Yaskawa INFORM job: KRIS1A.JBI

/JOB
//NAME KRIS1A
///FOLDERNAME X4
//POS
///NPOS 161,161,159,7,0,0
///TOOL 0
///POSTYPE PULSE
///PULSE
C00000=-15579,-90125,-112680,751,85832,86751
C00001=112118,-87719,-111704,295,86466,-7981
C00002=112804,-79721,-69104,72,64358,-7781
C00003=115139,-78813,-67219,-786,63674,-6908
C00004=115139,-78456,-66016,-789,63117,-6905
C00005=115139,-78780,-67104,-787,63620,-6908
C00006=114295,-93268,-73076,-493,59845,-7207
C00007=115346,-91281,-70266,-899,59147,-6796
C00008=115425,-89696,-69639,-926,59575,-6770
C00009=114013,-96528,-75756,-385,59817,-7318
C00010=112176,-79610,-68801,301,64230,-8016
C00011=111826,-77700,-66544,429,63826,-8147
C00012=111826,-77414,-65561,430,63368,-8149
C00013=112189,-78969,-67115,296,63524,-8012
C00014=110981,-94268,-73476,769,59585,-8491
C00015=111195,-90668,-69679,691,59097,-8412
C00016=111340,-88986,-69006,634,59545,-8354
C00017=110917,-95978,-76175,788,60368,-8510
C00018=98905,-94426,-81055,5125,64609,-12947
C00019=104248,-50126,-59827,871,84915,-31292
C00020=110771,-18155,-40833,-2727,97609,-44192
C00021=111360,-18636,-39123,-2768,96333,-43971
C00022=111360,-18738,-38396,-2766,95833,-43962
C00023=110217,-18316,-38887,-2668,96314,-44350
C00024=110620,-19725,-39043,-2697,95701,-44202
C00025=110670,-19738,-39055,-2703,95699,-44187
C00026=109565,-18053,-39144,-2612,96586,-44572
C00027=114086,43998,16856,-2992,94166,-43015
C00028=114053,43978,17325,-2992,93865,-43021
C00029=114053,43945,17976,-2992,93449,-43011
C00030=113191,44226,17588,-2916,93800,-43307
C00031=113191,44191,18270,-2913,93364,-43296
C00032=113504,44097,18169,-2941,93388,-43192
C00033=113191,44297,16563,-2919,94467,-43322
C00034=95546,58384,35854,30061,98673,-46154
C00035=95582,58774,36295,30055,98599,-46160
C00036=123577,27205,-10716,19125,86619,-21364
C00037=146491,35264,3200,11924,78186,-14764
C00038=139465,39684,6918,23498,85006,-10799
C00039=143221,41856,17232,31724,78736,-2144
C00040=143777,45964,21760,32091,77889,-1898
C00041=143777,45970,22332,32127,77590,-1984
C00042=143777,45964,21760,32091,77889,-1898
C00043=144048,47864,23803,32049,77548,-1889
C00044=143777,45964,21760,32091,77889,-1898
C00045=140515,27172,13,30557,79503,260
C00046=127712,47757,18303,22708,83382,-6719
C00047=131160,50524,19335,14874,81362,-8697
C00048=131524,51962,21137,14784,80938,-8621
C00049=131524,51834,22237,14811,80220,-8709
C00050=131524,51962,21137,14784,80938,-8621
C00051=131412,54587,24038,14832,80535,-8708
C00052=124540,58684,30159,20118,82239,-15737
C00053=124540,58684,30159,20118,82239,-15737
C00054=126244,67376,38231,22849,84013,-19503
C00055=125634,64122,36548,22992,83592,-19805
C00056=124813,61662,33823,22854,83980,-19602
C00057=136187,52210,23726,20634,82490,-16225
C00058=138691,53299,30320,37349,84215,-2442
C00059=138736,52471,34602,46175,82339,-1039
C00060=124737,44137,16346,44293,94212,-2593
C00061=119692,30389,-7142,25705,97127,-4865
C00062=118955,27408,-15020,17592,99243,-80195
C00063=125200,-2101,-32741,15880,81610,-85840
C00064=134088,-16964,-41109,182,70766,-85347
C00065=127415,46663,16862,1950,67717,-87809
C00066=121903,36391,497,16998,81593,-86950
C00067=125298,-36844,-66213,15778,84239,-85470
C00068=119205,-70443,-76936,24876,74885,-88203
C00069=118806,-67965,-71783,25211,73277,-88701
C00070=119684,40726,11380,24463,77277,-87514
C00071=126391,-52827,-68733,22124,76579,-85223
C00072=119612,-43604,-61782,23842,90714,-84840
C00073=150919,-31098,-53968,16672,84728,-75038
C00074=142912,-38104,-51044,32938,76311,-77903
C00075=131483,-69573,-74262,36162,79312,-81611
C00076=134129,-100468,-92829,36100,74575,-82089
C00077=-15579,-90125,-112680,751,85832,86751
C00078=-15579,-90125,-112680,751,85832,86751
C00079=-15579,-90125,-112677,751,85834,86750
C00080=-3695,-78746,-107796,-19987,71227,-76789
C00081=-15579,-90125,-112677,751,85834,86750
C00082=69723,-89114,-112269,359,86097,-2011
C00083=103224,-63598,-76709,4432,93708,-9007
C00084=100150,-62593,-71932,4790,91465,-10109
C00085=102335,-62307,-70304,4519,90489,-9417
C00086=102335,-62333,-69297,4519,89858,-9438
C00087=102335,-62306,-70332,4519,90507,-9413
C00088=99769,-80336,-79078,4826,86783,-10413
C00089=98266,-88378,-78396,6942,76534,-11334
C00090=98474,-87229,-77918,6891,76813,-11243
C00091=99558,-93232,-83375,6670,76995,-10858
C00092=70996,-48839,-62917,11636,90314,-19604
C00093=69525,-45287,-58669,11857,89748,-20153
C00094=69525,-45355,-57854,11856,89224,-20204
C00095=69525,-45284,-58714,11860,89779,-20150
C00096=64327,-57195,-66086,12620,89001,-21989
C00097=64937,-55938,-62941,12533,87648,-21918
C00098=65630,-54449,-62112,12434,87792,-21669
C00099=64207,-57448,-65984,12639,88833,-22049
C00100=106021,-71460,-78290,5261,84540,-8299
C00101=112603,-50924,-67434,3896,88035,39850
C00102=99785,-49787,-63878,14924,89163,36712
C00103=99827,-50120,-62714,14916,88297,36622
C00104=99827,-50195,-61812,14916,87722,36551
C00105=99827,-50144,-62447,14916,88126,36600
C00106=101735,-51128,-63015,14585,87637,37193
C00107=101608,-51204,-62348,14606,87222,37100
C00108=101075,-50939,-62194,14699,87359,36934
C00109=102139,-51368,-63677,14510,87842,37354
C00110=99650,-48435,-63078,14947,89385,36690
C00111=99972,-48773,-61841,14889,88425,36682
C00112=99972,-48836,-61171,14890,87997,36629
C00113=99984,-48651,-62050,14887,88610,36709
C00114=102057,-49715,-62671,14526,88085,37352
C00115=101809,-49682,-61617,14570,87514,37201
C00116=101235,-49486,-61523,14671,87658,37023
C00117=101817,-49661,-62901,14567,88291,37295
C00118=100331,-60546,-70178,19462,73070,35082
C00119=112110,-11200,-31080,-21080,73268,936
C00120=112400,17878,-3446,-21379,75013,1233
C00121=111590,19523,-1910,-21129,74714,991
C00122=111590,19505,-1171,-21171,74277,1069
C00123=111547,19542,-1905,-21114,74709,976
C00124=111586,21327,-236,-21132,74618,1008
C00125=111547,19542,-1905,-21114,74709,976
C00126=112862,2673,-16978,-21482,75612,1293
C00127=115448,-25762,-50567,-21911,81920,1062
C00128=115448,-26322,-48444,-21988,80436,1335
C00129=82803,-6073,-29763,-10236,73084,-8971
C00130=79384,-350,-31136,-8698,76436,-10385
C00131=79572,10395,-14436,-8965,71755,-9979
C00132=79534,10356,-13587,-8976,71217,-9951
C00133=79572,10395,-14436,-8965,71755,-9979
C00134=79918,12066,-12957,-9108,71739,-9858
C00135=79284,8995,-16143,-8832,72049,-10102
C00136=90478,36773,12863,-10350,74792,593
C00137=94157,33011,8641,-3718,74256,-1986
C00138=94889,36373,12557,5370,72876,-270
C00139=91513,44429,23385,15929,70108,-695
C00140=94206,50619,32489,25830,69108,-1135
C00141=99622,24209,5008,27862,67795,3286
C00142=101698,-3167,-21798,-5919,61845,73
C00143=117691,-82819,-72183,-15832,54407,7355
C00144=136102,-94056,-81974,-24248,59304,-21802
C00145=127300,-9107,-38878,-10715,73507,-75725
C00146=127883,-10256,-28747,-11426,66877,-74900
C00147=125820,57665,36060,-10904,61708,-75162
C00148=125724,45909,15983,-10333,67906,-75775
C00149=151418,-11051,-30715,-39158,77226,-70934
C00150=166637,-124928,-92814,-37840,63906,-58834
C00151=182097,-119423,-82240,-42095,69399,-53697
C00152=148901,-14656,-27686,-35717,72453,-69897
C00153=152618,-101160,-84187,-32865,63932,-65185
C00154=146642,-96347,-88741,-9688,84313,-74893
C00155=146358,-95495,-85194,-9676,82559,-74858
C00156=129145,-102178,-86219,-14985,78455,-80586
C00157=126274,-93471,-76691,-31678,80491,-81832
C00158=136204,-90113,-81071,-25794,88530,-79839
C00159=135637,-91176,-85093,-22103,89594,-80119
C00160=-3208,-93475,-86259,-2679,87523,-79016
BC00000=99,526410,1075081
BC00001=171737,515230,306420
BC00002=55459,454786,199131
BC00003=55459,454786,199131
BC00004=55459,454786,199131
BC00005=55459,454786,199131
BC00006=55459,454786,199131
BC00007=55459,454786,199131
BC00008=55459,454786,199131
BC00009=55459,454786,199131
BC00010=108304,454786,199131
BC00011=108304,454786,199131
BC00012=108304,454786,199131
BC00013=108304,454786,199131
BC00014=108304,454786,199131
BC00015=108304,454786,199131
BC00016=108304,454786,199131
BC00017=108304,454786,199131
BC00018=108304,454786,199131
BC00019=108304,454786,199131
BC00020=108304,454786,199131
BC00021=108304,454786,199131
BC00022=108304,454786,199131
BC00023=108304,454786,199131
BC00024=108304,454786,199131
BC00025=108304,454786,199131
BC00026=108304,454786,199131
BC00027=108304,440546,199131
BC00028=108304,440546,199131
BC00029=108304,440546,199131
BC00030=108304,440546,199131
BC00031=108304,440546,199131
BC00032=108304,440546,199130
BC00033=108304,440546,199131
BC00034=108304,440546,199131
BC00035=108304,440546,199131
BC00036=153886,383281,124194
BC00037=174583,383281,124194
BC00038=163957,383281,124194
BC00039=168122,383282,124193
BC00040=170139,383282,124190
BC00041=170139,383282,124190
BC00042=170139,383282,124190
BC00043=170139,383282,124190
BC00044=170139,383282,124190
BC00045=170139,383282,124190
BC00046=146661,383281,124193
BC00047=154148,383281,124194
BC00048=154148,383281,124194
BC00049=154148,383281,124194
BC00050=154148,383281,124194
BC00051=154148,383281,124194
BC00052=140502,383282,124191
BC00053=140502,383282,124191
BC00054=154149,383281,124191
BC00055=154149,383281,124191
BC00056=141565,383281,124189
BC00057=154149,383281,124188
BC00058=154152,383279,124187
BC00059=154149,383281,124191
BC00060=139202,383281,124191
BC00061=134656,383281,124191
BC00062=136731,381659,124191
BC00063=152069,383281,124191
BC00064=150142,383281,124191
BC00065=138256,383281,124191
BC00066=136697,383281,124191
BC00067=170077,383281,124191
BC00068=170077,446955,124191
BC00069=170077,446955,124191
BC00070=170077,446955,124191
BC00071=170077,446955,124191
BC00072=170077,446955,124191
BC00073=170077,446955,124191
BC00074=170077,446955,124191
BC00075=170077,446955,124191
BC00076=170077,446955,124191
BC00077=99,526410,1075081
BC00078=99,526410,1075081
BC00079=99,526409,1075080
BC00080=199448,515539,1075137
BC00081=141247,502779,337681
BC00082=222419,439021,164840
BC00083=279909,439021,164840
BC00084=279909,439021,164840
BC00085=279909,439021,164840
BC00086=279909,439021,164840
BC00087=279909,439021,164840
BC00088=279909,439021,164840
BC00089=279909,439021,164840
BC00090=279909,439021,164840
BC00091=279909,439021,164840
BC00092=279909,439021,164840
BC00093=279909,439021,164840
BC00094=279909,439021,164840
BC00095=279909,439021,164840
BC00096=279909,439021,164840
BC00097=279909,439021,164840
BC00098=279909,439021,164840
BC00099=279909,439021,164840
BC00100=279909,439021,164840
BC00101=279909,439021,164840
BC00102=279909,439021,164840
BC00103=279909,439021,164840
BC00104=279909,439021,164840
BC00105=279909,439021,164840
BC00106=279909,439021,164840
BC00107=279909,439021,164840
BC00108=279909,439021,164840
BC00109=279909,439021,164840
BC00110=279909,350395,164840
BC00111=279909,350395,164840
BC00112=279909,350395,164840
BC00113=279909,350395,164840
BC00114=279909,350395,164840
BC00115=279909,350395,164840
BC00116=279909,350395,164840
BC00117=279909,350395,164840
BC00118=279909,350395,164840
BC00119=279909,350395,164840
BC00120=279909,355371,164840
BC00121=279909,355371,164840
BC00122=279909,355371,164840
BC00123=279909,355371,164840
BC00124=279909,355371,164840
BC00125=279909,355371,164840
BC00126=279909,355371,164840
BC00127=279909,355371,164840
BC00128=279909,427919,164840
BC00129=247234,427919,164840
BC00130=278465,363509,138086
BC00131=278465,363509,138086
BC00132=278465,363509,138086
BC00133=278465,363509,138086
BC00134=278465,363509,138086
BC00135=278465,363509,138086
BC00136=302650,395853,164837
BC00137=311944,395852,164836
BC00138=309501,395853,164836
BC00139=296323,395854,164837
BC00140=301591,395854,164837
BC00141=326424,395853,164837
BC00142=326424,395853,164837
BC00143=326424,395853,164837
BC00144=326424,395853,164837
BC00145=326424,395853,164837
BC00146=326869,395161,164261
BC00147=326869,395161,164261
BC00148=326869,395161,164261
BC00149=326869,395161,164261
BC00150=326869,395161,164261
BC00151=326869,395161,164261
BC00152=326869,395161,164261
BC00153=326869,395161,164261
BC00154=326869,395161,164261
BC00155=326869,395161,164261
BC00156=326869,395161,164261
BC00157=326869,395161,164260
BC00158=326869,395161,164259
BC00159=326869,452441,213700
BC00160=87826,515074,1040939
EC00000=-798157,-183832
EC00001=-798154,-183834
EC00002=-798154,-183834
EC00003=-798154,-183834
EC00004=-798154,-183834
EC00005=-798154,-183834
EC00006=-798154,-183834
EC00007=-798154,-183834
EC00008=-798154,-183834
EC00009=-798154,-183834
EC00010=-798154,-183834
EC00011=-798154,-183834
EC00012=-798154,-183834
EC00013=-798154,-183834
EC00014=-798154,-183834
EC00015=-798154,-183834
EC00016=-798154,-183834
EC00017=-798154,-183834
EC00018=-798154,-183834
EC00019=-798154,-183834
EC00020=-798154,-183834
EC00021=-798154,-183834
EC00022=-798154,-183834
EC00023=-798154,-183834
EC00024=-798154,-183834
EC00025=-798154,-183834
EC00026=-798154,-183834
EC00027=-798154,-183834
EC00028=-798154,-183834
EC00029=-798154,-183834
EC00030=-798154,-183834
EC00031=-798154,-183834
EC00032=-798153,-183834
EC00033=-798154,-183834
EC00034=-798154,-183834
EC00035=-798154,-183834
EC00036=-798154,-183834
EC00037=-798154,-183834
EC00038=-798154,-183834
EC00039=-798153,-183835
EC00040=-798152,-183835
EC00041=-798152,-183835
EC00042=-798152,-183835
EC00043=-798152,-183835
EC00044=-798152,-183835
EC00045=-798152,-183835
EC00046=-798154,-183834
EC00047=-798154,-183834
EC00048=-798154,-183834
EC00049=-798154,-183834
EC00050=-798154,-183834
EC00051=-798154,-183834
EC00052=-798151,-183838
EC00053=-798151,-183838
EC00054=-798151,-183835
EC00055=-798151,-183835
EC00056=-798151,-183835
EC00057=-798153,-183834
EC00058=-798153,-183834
EC00059=-798153,-183834
EC00060=-798153,-183834
EC00061=-798153,-183834
EC00062=-798153,-183834
EC00063=-798153,-183834
EC00064=-798153,-183834
EC00065=-798153,-183834
EC00066=-798153,-183834
EC00067=-798153,-183834
EC00068=-798153,-183834
EC00069=-798153,-183834
EC00070=-798153,-183834
EC00071=-798153,-183834
EC00072=-798153,-183834
EC00073=-798153,-183834
EC00074=-798153,-183834
EC00075=-798157,-183832
EC00076=-93266,-194312
EC00077=-184298,-1289476
EC00078=-798157,-1296784
EC00079=-798157,-1296784
EC00080=-798156,-1296783
EC00081=-798156,-1296783
EC00082=-798156,-1296783
EC00083=-798156,-1296783
EC00084=-798156,-1296783
EC00085=-798156,-1296783
EC00086=-798156,-1296783
EC00087=-798156,-1296783
EC00088=-798156,-1296783
EC00089=-798156,-1296783
EC00090=-798156,-1296783
EC00091=-798156,-1296783
EC00092=-798156,-1296783
EC00093=-798156,-1296783
EC00094=-798156,-1296783
EC00095=-798156,-1296783
EC00096=-798156,-1296783
EC00097=-798156,-1296783
EC00098=-798156,-1296783
EC00099=-798156,-1296783
EC00100=-798156,-1296783
EC00101=-798156,-1296783
EC00102=-798156,-1296783
EC00103=-798156,-1296783
EC00104=-798156,-1296783
EC00105=-798156,-1296783
EC00106=-798156,-1296783
EC00107=-798156,-1296783
EC00108=-798156,-1296783
EC00109=-798156,-1296783
EC00110=-798156,-1296783
EC00111=-798156,-1296783
EC00112=-798156,-1296783
EC00113=-798156,-1296783
EC00114=-798156,-1296783
EC00115=-798156,-1296783
EC00116=-798156,-1296783
EC00117=-798156,-1296783
EC00118=-798156,-1296783
EC00119=-798156,-1296783
EC00120=-798156,-1296783
EC00121=-798156,-1296783
EC00122=-798156,-1296783
EC00123=-798156,-1296783
EC00124=-798156,-1296783
EC00125=-798156,-1296783
EC00126=-798156,-1296783
EC00127=-798156,-1296783
EC00128=-798156,-1296783
EC00129=-798156,-1296783
EC00130=-798156,-1296783
EC00131=-798156,-1296783
EC00132=-798156,-1296783
EC00133=-798156,-1296783
EC00134=-798155,-1296782
EC00135=-798154,-1296780
EC00136=-798153,-1296781
EC00137=-798154,-1296781
EC00138=-798154,-1296781
EC00139=-798155,-1296782
EC00140=-798155,-1296782
EC00141=-798155,-1296782
EC00142=-798155,-1296782
EC00143=-798155,-1296782
EC00144=-798155,-1296782
EC00145=-798155,-1296782
EC00146=-798155,-1296782
EC00147=-798155,-1296782
EC00148=-798155,-1296782
EC00149=-798155,-1296782
EC00150=-798155,-1296782
EC00151=-798155,-1296782
EC00152=-798155,-1296782
EC00153=-798155,-1296782
EC00154=-798155,-1296782
EC00155=-798154,-1296781
EC00156=-798154,-1296780
EC00157=-798154,-1296780
EC00158=-798154,-1287204
///POSTYPE BASE
///RECTAN
///RCONF 0,0,0,0,1,0,0,0,0,0,0,0,0,0,0,0,0,0,0,0,0,0,0,0
P00006=2.006,1.622,-0.565,0.0000,0.0000,0.0000
P00021=0.073,2.058,-0.109,0.0000,0.0000,0.0000
P00022=2.006,1.622,-0.565,0.0000,0.0000,0.0000
///RCONF 0,0,0,0,0,0,0,0,0,0,0,0,0,0,0,0,0,0,0,0,0,0,0,0
P00023=-2.957,-4.083,2.762,0.0000,0.0000,0.0000
P00024=-1.466,-0.226,-0.419,0.0000,0.0000,0.0000
P00025=3.643,0.007,-2.585,0.0000,0.0000,0.0000
P00026=2.644,0.055,-2.583,0.0000,0.0000,0.0000
//INST
///DATE 2024/11/13 16:42
///ATTR SC,RW
///GROUP1 RB1,BS1
///GROUP2 ST1
NOP
SFTOF3D
CALL JOB:CLEAN-R1_KM_NEW
MOVJ C00000 BC00000 VJ=100.00  +MOVJ EC00000 VJ=100.00
MOVJ C00001 BC00001 VJ=100.00  +MOVJ EC00001 VJ=100.00
MOVJ C00002 BC00002 VJ=100.00  +MOVJ EC00002 VJ=100.00
SMOVL C00003 BC00003 V=100.0  +MOVJ EC00003
SREFP 3 C00004 BC00004  +REFP EC00004
CALL JOB:SEARCH-R1-S13D
SET P023 P006
SFTON3D P023
SMOVL C00005 BC00005 V=133.3  +MOVJ EC00005
SMOVL C00006 BC00006 V=133.3  +MOVJ EC00006
SMOVL C00007 BC00007 V=133.3  +MOVJ EC00007
SREFP 3 C00008 BC00008  +REFP EC00008
CALL JOB:SEARCH-R1-S13D
SET P023 P006
SFTON3D P023
SMOVL C00009 BC00009 V=166.7  +MOVJ EC00009
SFTOF
SFTOF3D
SMOVL C00010 BC00010 V=250.0  +MOVJ EC00010
SMOVL C00011 BC00011 V=100.0  +MOVJ EC00011
SREFP 3 C00012 BC00012  +REFP EC00012
CALL JOB:SEARCH-R1-S13D
SET P024 P006
SFTON3D P024
SMOVL C00013 BC00013 V=133.3  +MOVJ EC00013
SMOVL C00014 BC00014 V=133.3  +MOVJ EC00014
SMOVL C00015 BC00015 V=133.3  +MOVJ EC00015
SREFP 3 C00016 BC00016  +REFP EC00016
CALL JOB:SEARCH-R1-S13D
SET P024 P006
SFTON3D P024
SMOVL C00017 BC00017 V=166.7  +MOVJ EC00017
SFTOF3D
MOVJ C00018 BC00018 VJ=100.00  +MOVJ EC00018 VJ=100.00
MOVJ C00019 BC00019 VJ=100.00  +MOVJ EC00019 VJ=100.00
MOVJ C00020 BC00020 VJ=100.00  +MOVJ EC00020 VJ=100.00
SMOVL C00021 BC00021 V=100.0  +MOVJ EC00021
SREFP 3 C00022 BC00022  +REFP EC00022
CALL JOB:SEARCH-R1-S13D
SET P025 P006
SFTON3D P025
SMOVL C00023 BC00023 V=100.0  +MOVJ EC00023
SMOVL C00024 BC00024 V=100.0  +MOVJ EC00024
SREFP 3 C00025 BC00025  +REFP EC00025
CALL JOB:SEARCH-R1-S13D
SET P025 P006
SFTON3D P025
SMOVL C00026 BC00026 V=100.0  +MOVJ EC00026
SFTOF3D
SFTOF
SMOVL C00027 BC00027 V=500.0  +MOVJ EC00027
SMOVL C00028 BC00028 V=100.0  +MOVJ EC00028
SREFP 3 C00029 BC00029  +REFP EC00029
CALL JOB:SEARCH-R1-S13D
SET P026 P006
SFTON3D P026
SMOVL C00030 BC00030 V=133.3  +MOVJ EC00030
SMOVL C00031 BC00031 V=100.0  +MOVJ EC00031
SREFP 3 C00032 BC00032  +REFP EC00032
CALL JOB:SEARCH-R1-S13D
SET P026 P006
SFTON3D P026
SMOVL C00033 BC00033 V=166.7  +MOVJ EC00033
SFTOF3D
SFTOF
SMOVL C00034 BC00034 V=500.0  +MOVJ EC00034
MOVJ C00035 BC00035 VJ=100.00  +MOVJ EC00035 VJ=100.00
MOVJ C00036 BC00036 VJ=100.00  +MOVJ EC00036 VJ=20.00
MOVJ C00037 BC00037 VJ=20.00  +MOVJ EC00037 VJ=20.00
MOVJ C00038 BC00038 VJ=20.00  +MOVJ EC00038 VJ=20.00
MOVJ C00039 BC00039 VJ=20.00  +MOVJ EC00039 VJ=20.00
SMOVL C00040 BC00040 V=100.0  +MOVJ EC00040
SREFP 3 C00041 BC00041  +REFP EC00041
CALL JOB:SEARCH-R1-S13D
SET P022 P006
SFTON3D P022
SMOVL C00042 BC00042 V=100.0  +MOVJ EC00042
SREFP 3 C00043 BC00043  +REFP EC00043
CALL JOB:SEARCH-R1-S13D
SET P022 P006
SFTON3D P022
SMOVL C00044 BC00044 V=100.0  +MOVJ EC00044
SFTOF3D
MOVL C00045 BC00045 V=500.0  +MOVJ EC00045 VJ=20.00
MOVL C00046 BC00046 V=500.0  +MOVJ EC00046 VJ=20.00
SMOVL C00047 BC00047 V=500.0  +MOVJ EC00047
SMOVL C00048 BC00048 V=100.0  +MOVJ EC00048
SREFP 3 C00049 BC00049  +REFP EC00049
CALL JOB:SEARCH-R1-S13D
SET P021 P006
SFTON3D P021
SMOVL C00050 BC00050 V=100.0  +MOVJ EC00050
SREFP 3 C00051 BC00051  +REFP EC00051
CALL JOB:SEARCH-R1-S13D
SET P021 P006
SFTON3D P021
SMOVL C00052 BC00052 V=100.0  +MOVJ EC00052
MACRO1 MJ#(0) ARGF21
SMOVL C00053 BC00053 V=250.0  +MOVJ EC00053
REFP 1 RB1 C00054 BC00054
REFP 2 RB1 C00055 BC00055
ARCON
SWVON WEV#(100)
SMOVL C00056 BC00056 V=8.3  +MOVJ EC00054
SFTON3D P022
SMOVL C00057 BC00057 V=8.3  +MOVJ EC00055
SMOVL C00058 BC00058 V=8.3  +MOVJ EC00056
SMOVL C00059 BC00059 V=8.3  +MOVJ EC00057
ARCOF
SWVOF
SFTOF
SFTOF3D
SMOVL C00060 BC00060 V=333.3  +MOVJ EC00058
SMOVL C00061 BC00061 V=666.7  +MOVJ EC00059
MOVJ C00062 BC00062 VJ=100.00  +MOVJ EC00060 VJ=20.00
MOVJ C00063 BC00063 VJ=70.00  +MOVJ EC00061 VJ=20.00
MACRO1 MJ#(0) ARGF20
SFTON3D P025
SMOVL C00064 BC00064 V=250.0  +MOVJ EC00062
ARCON
SFTON3D P026
SMOVL C00065 BC00065 V=7.5  +MOVJ EC00063
ARCOF
SWVOF
SFTOF3D
SFTOF
SMOVL C00066 BC00066 V=333.3  +MOVJ EC00064
SMOVL C00067 BC00067 V=666.7  +MOVJ EC00065
MACRO1 MJ#(0) ARGF14
SMOVL C00068 BC00068 V=500.0  +MOVJ EC00066
SFTON3D P025
SMOVL C00069 BC00069 V=166.7  +MOVJ EC00067
ARCON
SWVON WEV#(20)
SFTON3D P026
SMOVL C00070 BC00070 V=10.0  +MOVJ EC00068
ARCOF
SWVOF
SFTOF
SFTOF3D
SMOVL C00071 BC00071 V=333.3  +MOVJ EC00069
SFTON3D P024
SMOVL C00072 BC00072 V=166.7  +MOVJ EC00070
ARCON
SWVON WEV#(20)
SFTON3D P023
SMOVL C00073 BC00073 V=12.5  +MOVJ EC00071
SMOVL C00074 BC00074 V=12.5  +MOVJ EC00072
ARCOF
SWVOF
SFTOF
SFTOF3D
SMOVL C00075 BC00075 V=500.0  +MOVJ EC00073
SMOVL C00076 BC00076 V=1000.0  +MOVJ EC00074
MOVJ C00077 BC00077 VJ=100.00  +MOVJ EC00075 VJ=20.00
MOVJ C00078 BC00078 VJ=100.00  +MOVJ EC00076 VJ=100.00
MOVJ C00079 BC00079 VJ=100.00  +MOVJ EC00077 VJ=100.00
MOVJ C00080 BC00080 VJ=100.00  +MOVJ EC00078 VJ=100.00
'DRUGA STRONA
CALL JOB:CLEAN-R1_KM_NEW
MOVJ C00081 BC00081 VJ=100.00  +MOVJ EC00079 VJ=100.00
MOVJ C00082 BC00082 VJ=100.00  +MOVJ EC00080 VJ=100.00
MOVJ C00083 BC00083 VJ=100.00  +MOVJ EC00081 VJ=100.00
SFTOF3D
MOVJ C00084 BC00084 VJ=100.00  +MOVJ EC00082 VJ=100.00
SMOVL C00085 BC00085 V=166.7  +MOVJ EC00083
SREFP 3 C00086 BC00086  +REFP EC00084
CALL JOB:SEARCH-R1-S13D
SET P023 P006
SFTON3D P023
SMOVL C00087 BC00087 V=250.0  +MOVJ EC00085
SMOVL C00088 BC00088 V=250.0  +MOVJ EC00086
SMOVL C00089 BC00089 V=250.0  +MOVJ EC00087
SREFP 3 C00090 BC00090  +REFP EC00088
CALL JOB:SEARCH-R1-S13D
SET P023 P006
SFTON3D P023
SFTOF3D
SFTOF
SMOVL C00091 BC00091 V=250.0  +MOVJ EC00089
SMOVL C00092 BC00092 V=250.0  +MOVJ EC00090
SMOVL C00093 BC00093 V=250.0  +MOVJ EC00091
SREFP 3 C00094 BC00094  +REFP EC00092
CALL JOB:SEARCH-R1-S13D
SET P024 P006
SFTON3D P024
SMOVL C00095 BC00095 V=250.0  +MOVJ EC00093
SMOVL C00096 BC00096 V=250.0  +MOVJ EC00094
SMOVL C00097 BC00097 V=250.0  +MOVJ EC00095
SREFP 3 C00098 BC00098  +REFP EC00096
CALL JOB:SEARCH-R1-S13D
SET P024 P006
SFTON3D P024
SFTOF3D
SMOVL C00099 BC00099 V=250.0  +MOVJ EC00097
MOVJ C00100 BC00100 VJ=100.00  +MOVJ EC00098 VJ=100.00
MOVJ C00101 BC00101 VJ=100.00  +MOVJ EC00099 VJ=100.00
MOVJ C00102 BC00102 VJ=100.00  +MOVJ EC00100 VJ=100.00
SMOVL C00103 BC00103 V=250.0  +MOVJ EC00101
SREFP 3 C00104 BC00104  +REFP EC00102
CALL JOB:SEARCH-R1-S13D
SET P025 P006
SFTON3D P025
SMOVL C00105 BC00105 V=250.0  +MOVJ EC00103
SMOVL C00106 BC00106 V=250.0  +MOVJ EC00104
SMOVL C00107 BC00107 V=100.0  +MOVJ EC00105
SREFP 3 C00108 BC00108  +REFP EC00106
CALL JOB:SEARCH-R1-S13D
SET P025 P006
SFTON3D P025
SFTOF3D
SMOVL C00109 BC00109 V=100.0  +MOVJ EC00107
SMOVL C00110 BC00110 V=333.3  +MOVJ EC00108
SMOVL C00111 BC00111 V=250.0  +MOVJ EC00109
SREFP 3 C00112 BC00112  +REFP EC00110
CALL JOB:SEARCH-R1-S13D
SET P026 P006
SFTON3D P026
SMOVL C00113 BC00113 V=250.0  +MOVJ EC00111
SMOVL C00114 BC00114 V=250.0  +MOVJ EC00112
SMOVL C00115 BC00115 V=100.0  +MOVJ EC00113
SREFP 3 C00116 BC00116  +REFP EC00114
CALL JOB:SEARCH-R1-S13D
SET P026 P006
SFTON3D P026
SFTOF3D
SMOVL C00117 BC00117 V=250.0  +MOVJ EC00115
SMOVL C00118 BC00118 V=333.3  +MOVJ EC00116
MOVJ C00119 BC00119 VJ=20.00  +MOVJ EC00117 VJ=20.00
MOVJ C00120 BC00120 VJ=20.00  +MOVJ EC00118 VJ=20.00
SMOVL C00121 BC00121 V=250.0  +MOVJ EC00119
SREFP 3 C00122 BC00122  +REFP EC00120
CALL JOB:SEARCH-R1-S13D
SET P021 P006
SFTON3D P021
SMOVL C00123 BC00123 V=250.0  +MOVJ EC00121
SREFP 3 C00124 BC00124  +REFP EC00122
CALL JOB:SEARCH-R1-S13D
SET P021 P006
SFTON3D P021
SFTOF3D
SMOVL C00125 BC00125 V=250.0  +MOVJ EC00123
MOVL C00126 BC00126 V=250.0  +MOVJ EC00124 VJ=20.00
MOVL C00127 BC00127 V=333.3  +MOVJ EC00125 VJ=20.00
SMOVL C00128 BC00128 V=1000.0  +MOVJ EC00126
SMOVL C00129 BC00129 V=1000.0  +MOVJ EC00127
SMOVL C00130 BC00130 V=250.0  +MOVJ EC00128
SMOVL C00131 BC00131 V=250.0  +MOVJ EC00129
SREFP 3 C00132 BC00132  +REFP EC00130
CALL JOB:SEARCH-R1-S13D
SET P022 P006
SFTON3D P022
SMOVL C00133 BC00133 V=250.0  +MOVJ EC00131
SREFP 3 C00134 BC00134  +REFP EC00132
CALL JOB:SEARCH-R1-S13D
SET P022 P006
SFTOF3D
SMOVL C00135 BC00135 V=250.0  +MOVJ EC00133
MACRO1 MJ#(0) ARGF21
SFTON3D P022
SMOVL C00136 BC00136 V=250.0  +MOVJ EC00134
ARCON
SWVON WEV#(100)
SMOVL C00137 BC00137 V=8.3  +MOVJ EC00135
SMOVL C00138 BC00138 V=8.3  +MOVJ EC00136
SFTON3D P021
SMOVL C00139 BC00139 V=8.3  +MOVJ EC00137
SMOVL C00140 BC00140 V=8.3  +MOVJ EC00138
ARCOF
SFTOF3D
SWVOF
SMOVL C00141 BC00141 V=250.0  +MOVJ EC00139
SMOVL C00142 BC00142 V=500.0  +MOVJ EC00140
MOVJ C00143 BC00143 VJ=50.00  +MOVJ EC00141 VJ=20.00
MOVJ C00144 BC00144 VJ=100.00  +MOVJ EC00142 VJ=20.00
MOVJ C00145 BC00145 VJ=40.00  +MOVJ EC00143 VJ=20.00
MACRO1 MJ#(0) ARGF20
SFTON3D P025
SMOVL C00146 BC00146 V=133.3 PL=0  +MOVJ EC00144
ARCON
SFTON3D P026
SMOVL C00147 BC00147 V=6.7  +MOVJ EC00145
ARCOF
SWVOF
SFTOF3D
SMOVL C00148 BC00148 V=250.0  +MOVJ EC00146
SMOVL C00149 BC00149 V=500.0  +MOVJ EC00147
MACRO1 MJ#(0) ARGF14
SFTOF3D
SMOVL C00150 BC00150 V=500.0  +MOVJ EC00148
SFTOF
SFTON3D P025
SMOVL C00151 BC00151 V=250.0  +MOVJ EC00149
ARCON
SWVON WEV#(20)
SFTON3D P026
SMOVL C00152 BC00152 V=10.0  +MOVJ EC00150
ARCOF
SWVOF
SFTOF3D
SMOVL C00153 BC00153 V=333.3  +MOVJ EC00151
MOVL C00154 BC00154 V=250.0  +MOVJ EC00152 VJ=100.00
SFTON3D P023
SMOVL C00155 BC00155 V=250.0  +MOVJ EC00153
ARCON
SWVON WEV#(20)
SFTON3D P024
SMOVL C00156 BC00156 V=11.7  +MOVJ EC00154
SMOVL C00157 BC00157 V=11.7  +MOVJ EC00155
ARCOF
SWVOF
SFTOF
SMOVL C00158 BC00158 V=250.0  +MOVJ EC00156
MOVJ C00159 BC00159 VJ=100.00  +MOVJ EC00157 VJ=20.00
MOVJ C00160 BC00160 VJ=100.00  +MOVJ EC00158 VJ=100.00
END
